// TIA Portal V19 export
DATA_BLOCK "DB_Techno"   // DB45
{ S7_Optimized_Access := 'FALSE' }
AUTHOR : RE
// stored: AutoNumber false
   VAR RETAIN
      DATEN_gueltig : Bool := FALSE;   // bit 0.0 rest vom Byte reserviert set:PC reset:SPS
      WT_NR_lng : DInt := 0;   // Warenträgernummer lang
      WT_NR_kurz : Byte := 16#00;   // wenn 0, dann Neuaufgabe eines WT
      STAND_NR : Byte := 16#00;   // wenn 0, dann Technologieänderung
      Oberflaeche : Real := 1.0;
      Prioritaet : Byte := 16#00;   // priorisierter WT Bit 12.0==1
      res : Bool := FALSE;
      res1 : Bool := FALSE;
      res2 : Bool := FALSE;
      res3 : Bool := FALSE;
      res4 : Bool := FALSE;
      res5 : Bool := FALSE;
      res6 : Bool := FALSE;
      res7 : Bool := FALSE;
      Korb_Nr : USInt;   // Korbnummer (fest)
      resByte : USInt;   // aktuelle Position
      Technologie : Int := 0;   // Technologie Code
      resW1 : Int := 0;
      resW2 : Int := 0;
      ParaByte : Byte := 16#00;   // Parameterbyte (inf. langsam Heben 22.1/Senken 22.0)
      WT_Typ : Byte := 16#00;   // Warenträgertyp B#16#11=KS, 12=LS, B#16#2x=GO
      resW3 : Int := 0;
      resD : DInt := 0;
      resD1 : DInt := 0;
      resD2 : DInt := 0;
      KorrPend : Real := 0.0;
      KorrATZ : Real := 0.0;
      Beginn_Daten : Int := 78;   // * Beginn des Technologiedatenblocks
      Ende_Daten : Int := 440;   // * Ende des Technologiedatenblocks
      resDW : DInt := 0;
      resDW1 : DInt := 0;
      resW4 : Int := 0;
      resW6 : Int := 0;
      AnzPendHub : Byte := 16#00;   // Anzahl Mehrfachhub
      WT_Kennung : Byte := 16#00;
      Speed_Up : Int := 0;   // Geschwindigkeitsbegrenzung Heben
      Speed_Dn : Int := 0;   // Geschwindigkeitsbegrenzung Senken
      Speed_Fahrt : Int := 0;   // Geschwindigkeitsbegrenzung Fahren (Ware)
      resI1 : Int := 0;
      resI2 : Int := 0;
      resI3 : Int := 0;
      resI4 : Int := 0;
      "Name" : String[100];
      stBefehle : Array[1..20] of Struct   // * bei Änderung anpassen
         Kennung : Byte;   // Befehlskennung
         FirstPos1 : Byte;   // erste Position, die angefahren werden kann
         Grpleng1 : Byte;   // Gruppenbad Länge
         FirstPos2 : Byte;
         Grpleng2 : Byte;
         Merker : Byte;
         Param_Ptr : Int;   // Pointer für Parameter
      END_STRUCT;
      stParam_Bereich : Array[1..100] of Byte;   // * bei Änderung oder Adressverschiebung anpassen
   END_VAR
BEGIN
   stBefehle[1..10].Kennung := 16#00;
   stBefehle[1..10].FirstPos1 := 16#00;
   stBefehle[1..10].Grpleng1 := 16#00;
   stBefehle[1..10].FirstPos2 := 16#00;
   stBefehle[1..10].Grpleng2 := 16#00;
   stBefehle[1..10].Merker := 16#00;
   stBefehle[1..10].Param_Ptr := 0;
   stParam_Bereich[1..100] := 16#00;
END_DATA_BLOCK
